FUNCTION_BLOCK FB_EM_Work EXTENDS FB_PackML_BaseModule
VAR
	// Submodules
	
	// Components
	
	// Module Data
	// --Param
	// --Recipe
	// --HMI
	
	// Alarms
	
	// Other I/O
	
	// Miscellaneous
	
END_VAR

METHOD PROTECTED Aborted
VAR_INPUT
END_VAR
END_METHOD

METHOD PROTECTED Aborting
VAR_INPUT
END_VAR
CASE _CurrentMode OF
	E_PMLUnitMode.ePMLUnitMode_Production:
        CASE DescendantSequenceState OF
			0:
				NoStateTasksToComplete := FALSE;
				DescendantSequenceState := DescendantSequenceState + 10;
			10:
				StateTasksComplete := TRUE;
		END_CASE
		
	E_PMLUnitMode.ePMLUnitMode_Manual, E_PMLUnitMode.ePMLUnitMode_Maintenance:
        ;	
END_CASE

// Call Super
SUPER^.Aborting();
END_METHOD

METHOD PROTECTED Clearing
VAR_INPUT
END_VAR
CASE _CurrentMode OF
	E_PMLUnitMode.ePMLUnitMode_Production:
        CASE DescendantSequenceState OF
			0:
				NoStateTasksToComplete := FALSE;
				DescendantSequenceState := DescendantSequenceState + 10;
			10:
				StateTasksComplete := TRUE;
		END_CASE
		
	E_PMLUnitMode.ePMLUnitMode_Manual, E_PMLUnitMode.ePMLUnitMode_Maintenance:
        ;	
END_CASE

// Call Super
SUPER^.Clearing();
END_METHOD

METHOD PROTECTED Complete
VAR_INPUT
END_VAR
END_METHOD

//! @summary Initializes event function blocks using this module's name
METHOD PROTECTED CreateEvents

//! @description This method is called by <c>Initialize()</c> as required
// Add your event creation here

// Super call to base
SUPER^.CreateEvents();
END_METHOD

METHOD CyclicLogic
VAR_INPUT
END_VAR
IF NOT _InitComplete THEN
    _InitComplete := Initialize();
    RETURN;
END_IF

SUPER^.CyclicLogic();
END_METHOD

METHOD PROTECTED Execute
VAR_INPUT
END_VAR
CASE _CurrentMode OF
	E_PMLUnitMode.ePMLUnitMode_Production:
        CASE DescendantSequenceState OF
			0:
				DescendantSequenceState := DescendantSequenceState + 10;
			10:
				;
		END_CASE
		
	E_PMLUnitMode.ePMLUnitMode_Manual, E_PMLUnitMode.ePMLUnitMode_Maintenance:
        ;	
END_CASE
END_METHOD

METHOD PROTECTED Held
VAR_INPUT
END_VAR
END_METHOD

METHOD PROTECTED Holding
VAR_INPUT
END_VAR
CASE _CurrentMode OF
	E_PMLUnitMode.ePMLUnitMode_Production:
        CASE DescendantSequenceState OF
			0:
				NoStateTasksToComplete := FALSE;
				DescendantSequenceState := DescendantSequenceState + 10;
			10:
				StateTasksComplete := TRUE;
		END_CASE
		
	E_PMLUnitMode.ePMLUnitMode_Manual, E_PMLUnitMode.ePMLUnitMode_Maintenance:
        ;	
END_CASE

// Call Super
SUPER^.Holding();
END_METHOD

METHOD PROTECTED Idle
VAR_INPUT
END_VAR
END_METHOD

//! @summary Basic module initialization logic
METHOD PROTECTED Initialize : BOOL;
VAR
	i						 : UDINT;
	varInfo					 : __SYSTEM.VAR_INFO;
	AllSubUnitsInitialized	 : BOOL := TRUE;
	AllComponentsInitialized : BOOL := TRUE;
END_VAR

//! @description This method is called by <c>CyclicLogic()</c> as required
Initialize := FALSE;
CASE DescendantSequenceState OF
    0: // Initialize
        _LogModeChanges         := FALSE;
        _LogStateChanges        := FALSE;
        DescendantSequenceState := DescendantSequenceState + 10;
	
	10: // Register Submodules
		//RegisterSubmodule(submodule);
		DescendantSequenceState := DescendantSequenceState + 10;
    20: // Register Components
		//RegisterComponent(component);
        DescendantSequenceState := DescendantSequenceState + 10;
    30: // Call the Super
        IF SUPER^.Initialize() THEN
            DescendantSequenceState := DescendantSequenceState + 10;
        END_IF
    40:
        Initialize := TRUE;
END_CASE
END_METHOD

METHOD PROTECTED Resetting
VAR_INPUT
END_VAR
CASE _CurrentMode OF
	E_PMLUnitMode.ePMLUnitMode_Production:
        CASE DescendantSequenceState OF
			0:
				NoStateTasksToComplete := FALSE;
				DescendantSequenceState := DescendantSequenceState + 10;
			10:
				StateTasksComplete := TRUE;
		END_CASE
		
	E_PMLUnitMode.ePMLUnitMode_Manual, E_PMLUnitMode.ePMLUnitMode_Maintenance:
        ;	
END_CASE

// Call Super
SUPER^.Resetting();
END_METHOD

METHOD PROTECTED Starting
VAR_INPUT
END_VAR
CASE _CurrentMode OF
	E_PMLUnitMode.ePMLUnitMode_Production:
        CASE DescendantSequenceState OF
			0:
				NoStateTasksToComplete := FALSE;
				DescendantSequenceState := DescendantSequenceState + 10;
			10:
				StateTasksComplete := TRUE;
		END_CASE
		
	E_PMLUnitMode.ePMLUnitMode_Manual, E_PMLUnitMode.ePMLUnitMode_Maintenance:
        ;	
END_CASE

// Call Super
SUPER^.Starting();
END_METHOD

METHOD PROTECTED Stopped
VAR_INPUT
END_VAR
END_METHOD

METHOD PROTECTED Stopping
VAR_INPUT
END_VAR
CASE _CurrentMode OF
	E_PMLUnitMode.ePMLUnitMode_Production:
        CASE DescendantSequenceState OF
			0:
				NoStateTasksToComplete := FALSE;
				DescendantSequenceState := DescendantSequenceState + 10;
			10:
				StateTasksComplete := TRUE;
		END_CASE
		
	E_PMLUnitMode.ePMLUnitMode_Manual, E_PMLUnitMode.ePMLUnitMode_Maintenance:
        ;	
END_CASE

// Call Super
SUPER^.Stopping();
END_METHOD

METHOD PROTECTED Suspended
VAR_INPUT
END_VAR
END_METHOD

METHOD PROTECTED Suspending
VAR_INPUT
END_VAR
CASE _CurrentMode OF
	E_PMLUnitMode.ePMLUnitMode_Production:
        CASE DescendantSequenceState OF
			0:
				NoStateTasksToComplete := FALSE;
				DescendantSequenceState := DescendantSequenceState + 10;
			10:
				StateTasksComplete := TRUE;
		END_CASE
		
	E_PMLUnitMode.ePMLUnitMode_Manual, E_PMLUnitMode.ePMLUnitMode_Maintenance:
        ;	
END_CASE

// Call Super
SUPER^.Suspending();
END_METHOD

METHOD PROTECTED Undefined
VAR_INPUT
END_VAR
END_METHOD

METHOD PROTECTED Unholding
VAR_INPUT
END_VAR
CASE _CurrentMode OF
	E_PMLUnitMode.ePMLUnitMode_Production:
        CASE DescendantSequenceState OF
			0:
				NoStateTasksToComplete := FALSE;
				DescendantSequenceState := DescendantSequenceState + 10;
			10:
				StateTasksComplete := TRUE;
		END_CASE
		
	E_PMLUnitMode.ePMLUnitMode_Manual, E_PMLUnitMode.ePMLUnitMode_Maintenance:
        ;	
END_CASE

// Call Super
SUPER^.Unholding();
END_METHOD

METHOD PROTECTED Unsuspending
VAR_INPUT
END_VAR
CASE _CurrentMode OF
	E_PMLUnitMode.ePMLUnitMode_Production:
        CASE DescendantSequenceState OF
			0:
				NoStateTasksToComplete := FALSE;
				DescendantSequenceState := DescendantSequenceState + 10;
			10:
				StateTasksComplete := TRUE;
		END_CASE
		
	E_PMLUnitMode.ePMLUnitMode_Manual, E_PMLUnitMode.ePMLUnitMode_Maintenance:
        ;	
END_CASE

// Call Super
SUPER^.Unsuspending();
END_METHOD

END_FUNCTION_BLOCK

(* stored: Version 1.1.0.1, ProductVersion 3.1.4024.12
   POU FB_EM_Work: Id {2ee5a866-b8eb-4e03-bc9e-c8be5ccee6d1}, SpecialFunc None
   Folder PackML: Id {6860c64a-d420-4a60-ac99-994d50770e67}
   Folder Acting States: Id {6e9e71cc-2e2a-404f-b2c8-48ff6cd0d1ed}
   Folder Waiting States: Id {cea085db-4679-4437-ad86-983701ec994d}
   Folder REFs: Id {8c42d4bf-fe40-4477-bde9-91826866164c}
   Method Aborted: Id {e8c3e360-0369-4864-9e80-993078c4e2cd}
   Method Aborting: Id {67160e95-7f39-46a7-9f91-3c5e2867d3df}
   Method Clearing: Id {604446e8-e37a-4e0e-a514-588a019bc1f2}
   Method Complete: Id {817ea939-88f0-41b4-a596-2b3f0d54f2e2}
   Method CreateEvents: Id {2ed811a8-478d-40b7-bf50-1f2a8f9af363}
   Method CyclicLogic: Id {a51d14b1-6c76-4901-92ca-9c7862e36047}
   Method Execute: Id {7a75d2a7-3bb4-4632-993d-33175f999cfd}
   Method Held: Id {43f5cec9-043a-41c4-b2d5-15a9fbc0ce34}
   Method Holding: Id {53d3b2ae-b1fa-45cf-a857-91c07cabfe94}
   Method Idle: Id {372ab538-a41a-45c9-8379-1cf30e5a4791}
   Method Initialize: Id {52ebd532-0cc8-49f4-bfb7-40197ee9bd5c}
   Method Resetting: Id {ae1b2d3a-b695-4006-9bc3-a8df4f28f741}
   Method Starting: Id {073393b8-c029-4c92-b746-59982aae1455}
   Method Stopped: Id {a7e85a21-d654-430d-87d0-b19f5e51c29e}
   Method Stopping: Id {1acaf942-5877-4658-a286-036e1477e9e5}
   Method Suspended: Id {0ebfafe7-4c6c-4e00-bb66-c2f0bfba56e5}
   Method Suspending: Id {ba71f435-1bd1-46cf-a491-40b61212bfc7}
   Method Undefined: Id {ce65f851-922e-4983-9161-a774acef8f1a}
   Method Unholding: Id {bb260919-c599-4e40-988f-9049b175db6f}
   Method Unsuspending: Id {716c933f-3905-498b-bed4-057b361cdd71} *)
